INTERFACE I_StoppedCommands

METHOD PUBLIC Reset
END_METHOD

END_INTERFACE

(* stored: Version 1.1.0.1, ProductVersion 3.1.4026.6
   Itf I_StoppedCommands: Id {1719d416-8cac-0ada-1b61-0b25b7a48bba}
   Method Reset: Id {feb743ed-94f8-07ef-3bbd-fcb7c4d31c83} *)
